TYPE Inbound_roller :
STRUCT
	roller : ARRAY[0..1] OF Roller;
	photo_sensor	: ARRAY[0..1] OF BOOL;//[1] light curtain mute
	mcAxis			: FB_MotionAxis_MC;
	st_mcAxis 		: ST_MotionAxis_MC;
	AxisRef			: AXIS_REF;
END_STRUCT
END_TYPE

(* stored: Version 1.1.0.1, ProductVersion 3.1.4024.12
   DUT Inbound_roller: Id {2a1bb7a1-a33e-4948-ae85-a9dd17bdc16c} *)
